// TIA Portal V16 export
// export: Created 2021-03-05T14:22:12.6455613Z, ExportSetting WithDefaults, DisplayName Totally Integrated Automation Portal, DisplayVersion V16, DisplayName TIA Portal Version Control Interface, DisplayVersion V16, DisplayName TIA Portal Openness, DisplayVersion V16, DisplayName SINAMICS Startdrive Advanced, DisplayVersion V16, DisplayName SINAMICS Startdrive G130, G150, S120, S150, SINAMICS MV, S210, DisplayVersion V16, DisplayName SINAMICS Startdrive G110M, G120, G120C, G120D, G120P, DisplayVersion V16, DisplayName STEP 7 Professional, DisplayVersion V16, DisplayName STEP 7 Safety, DisplayVersion V16, DisplayName WinCC Professional, DisplayVersion V16
FUNCTION_BLOCK "fbShelfFertigation"   // FB5, LAD
{ S7_Optimized_Access := 'TRUE' }
VERSION : 0.1
// stored: AutoNumber true, IsIECCheckEnabled false, IsRetainMemResEnabled false, MemoryReserve 100, SetENOAutomatically false, UDAEnableTagReadback false
   VAR_INPUT
      activeShelf : Int;
      shelfNumber : Int;
      ReservoirLevel : Real;
      RunMode : Int;
   END_VAR
   VAR_OUTPUT
      arrDQ : Array[1.."MAX_DQ_SHELF"] of Bool;
      DQ AT arrDQ : "udtShelfDQ";
   END_VAR
   VAR RETAIN
      Controls : Struct
         Flood_Duration : LInt := 5;   // Minutes
         Flood_Interval : Int := 288;   // Minutes
         Last_Flood : Date_And_Time := DT#2015-01-01-00:00:00;
         FillCommand : Bool;
         DrainCommand : Bool;
         WaterVolumeLimit : Real := 18.0;   // Gallons. Max amount of water a shelf can safely hold. If this limit is reached there might be a problem with the level switch (see overfill alarm)
         TON_Soak : TON_TIME;
         TON_Drain : TON_TIME;
      END_STRUCT;
      Status : Struct
         Active : Bool;
         Filling : Bool;
         Soaking : Bool;
         Soaking_Finished : Bool;
         Draining : Bool;
         Finished : Bool;
         OverfillAlarm : Bool;
      END_STRUCT;
   END_VAR
   VAR
      DQ_Fill_Solenoid : "udtDigitalOutput";
      DQ_Drain_Solenoid : "udtDigitalOutput";
      DI_Level_Switch : "udtDigitalInput";
   END_VAR
   VAR RETAIN
      iNextStep : UInt := 3;
   END_VAR
   VAR
      InitialReservoirLevel : Real;
   END_VAR
   VAR_TEMP
      ReservoirDelta : Real;
      i : Int;
      current_date_time : Date_And_Time;
      retval : Int;
      td_diff : Time;
      minutes_diff : LInt;
      current_date : LDT;
      current_time : LTime_Of_Day;
      shelf_last_date : LDT;
      day_diff : LTime;
      shelf_last_time : LTime_Of_Day;
      flood_time : Time;
      active_shelves : Int;
      j : Int;
   END_VAR
   VAR CONSTANT
      drain_time : Time := T#300S;
      eStep_Fill : UInt;
      eStep_Soak : UInt := 1;
      eStep_Drain : UInt := 2;
      eStep_Done : UInt := 3;
   END_VAR
BEGIN

REGION Network 1 (SCL): Flood, soak, drain routine

   IF #RunMode = 0 THEN
       #iNextStep := #eStep_Done;

   ELSIF #RunMode = 2 THEN
       IF #iNextStep = #eStep_Done THEN
           IF #activeShelf <> #shelfNumber THEN
               #iNextStep := #eStep_Done;
           ELSE
               #iNextStep := #eStep_Fill;
               // set initial reservoir level for delta calculation below to prevent overfilling shelf
               #InitialReservoirLevel := #ReservoirLevel;
           END_IF;
       END_IF;

       IF NOT #Status.Active THEN
           #iNextStep := #eStep_Done;
       END_IF;

       REGION 0: fill

           //stop filling if reservoir drops 70L or more, set a level switch alarm for shelf
           #ReservoirDelta := #InitialReservoirLevel - #ReservoirLevel;

           //IF #ReservoirDelta >= #Controls.WaterVolumeLimit THEN
               //#Status.Filling := 0;
               //#Controls.FillCommand := FALSE;
               //#iNextStep := #eStep_Soak;
               //#Status.OverfillAlarm := True;
           //END_IF;

           IF #iNextStep = #eStep_Fill THEN
               // while the level switch is in its normal position, fill 
               IF (#DI_Level_Switch.bStatus = #DI_Level_Switch.bNormalPosition) THEN
                   #Status.Filling := 1;
                   #Controls.FillCommand := True;
               ELSIF (#DI_Level_Switch.bStatus <> #DI_Level_Switch.bNormalPosition) THEN
                   #Status.Filling := 0;
                   #Controls.FillCommand := FALSE;
                   #iNextStep := #eStep_Soak;
               END_IF;
           END_IF;
       END_REGION


       REGION 1: Soak
           #flood_time := LINT_TO_TIME(#Controls.Flood_Duration * 60000);
           #Controls.TON_Soak(IN := (#iNextStep = #eStep_Soak),
                              PT := #flood_time,
                              Q => #Status.Soaking_Finished);

           IF #iNextStep = #eStep_Soak THEN
               #Status.Soaking := 1;
               IF #Status.Soaking_Finished THEN
                   #Status.Soaking := 0; //reset flood TON
                   #iNextStep := #eStep_Drain;
               END_IF;
           END_IF;
       END_REGION


       REGION 2: drain
           #Controls.TON_Drain(IN := (#iNextStep = #eStep_Drain),
                               PT := #drain_time,
                               Q => #Status.Finished);

           IF #iNextStep = #eStep_Drain THEN
               IF #activeShelf = #shelfNumber THEN
                   #Status.Draining := 1;
                   //open drain solenoid
                   #Controls.DrainCommand := TRUE;

                   IF #Status.Finished THEN
                       //close drain solenoid
                       #Controls.DrainCommand := FALSE;
                       #Status.Draining := 0; // reset drain TON
                       #Status.Soaking_Finished := 0;
                       #retval := RD_LOC_T(#Controls.Last_Flood);
                       #iNextStep := #eStep_Done;
                   END_IF;
               END_IF;

           END_IF;
       END_REGION

   ELSIF #RunMode = 3 THEN //discharge

       // TODO REMOVE THIS CONDITIONAL INCLUDING iNextStep ELSE CLAUSE
       //IF #Status.Active AND #activeShelf = #shelfNumber THEN
           // drain active shelf while rack is in discharge mode 
           #Controls.FillCommand := FALSE;
           #Controls.DrainCommand := TRUE;
           #Status.Filling := 0;
           #Status.Soaking := 0;
           #Status.Soaking_Finished := 0;
           #Status.Draining := 1;
           #iNextStep := #eStep_Drain; // this keeps us in drain mode untill RunMode is changed
       //ELSE
          // #iNextStep := #eStep_Done;
       //END_IF;

   END_IF;

   REGION 3: Done
       IF #iNextStep = #eStep_Done THEN
           // set these here in case shelf deactivated mid-operation
           #Controls.FillCommand := FALSE;
           #Controls.DrainCommand := FALSE;
           IF (#Status.Filling OR #Status.Soaking OR #Status.Draining) AND #activeShelf = #shelfNumber THEN
               #Status.Finished := 1;
           END_IF;
           #Status.Filling := 0;
           #Status.Soaking := 0;
           #Status.Soaking_Finished := 0;
           #Status.Draining := 0;

       END_IF;

   END_REGION
END_REGION

REGION Network 2 (SCL): write DQ outputs
   #DQ.Q_Fill_Solenoid := "fcDigitalOutput"(bInAutoVal := #Controls.FillCommand, InOutUdt := #DQ_Fill_Solenoid);
   #DQ.Q_Drain_Solenoid := "fcDigitalOutput"(bInAutoVal := #Controls.DrainCommand, InOutUdt := #DQ_Drain_Solenoid);
END_REGION
END_FUNCTION_BLOCK
